(* IEC 61131-3 sources: programs/VI-54/VI-54_20171205/VI-54_20171205/Stations/Screen/LseClass170718/Class/TCPComSend, 1 file *)

(* ---- TCPComSend.st ---- *)
(*!
<Class
	Name               = "TCPComSend"
	Revision           = "1.2"
	RealtimeTask       = "false"
	CyclicTask         = "true"
	BackgroundTask     = "true"
	Sigmatek           = "true"
	OSInterface        = "false"
	HighPriority       = "false"
	Automatic          = "false"
	UpdateMode         = "Prescan"
	SharedCommandTable = "true"
	Objectsize         = "(600,360)"
	Comment            = "Sending data via communication class.">
	<Channels>
		<Server Name="ClassSvr" Visualized="false" Initialize="false" WriteProtected="false" Retentive="false"/>
		<Server Name="ID_Destination" Visualized="false" Initialize="true" WriteProtected="true" Retentive="false"/>
		<Server Name="ID_Source" Visualized="false" Initialize="true" WriteProtected="true" Retentive="false"/>
		<Server Name="sSendCnt" Visualized="false" Initialize="false" WriteProtected="false" Retentive="false" Comment="Counter for sended data blocks."/>
		<Server Name="sSendErr" Visualized="false" Initialize="false" WriteProtected="false" Retentive="false" Comment="Counter for send errors."/>
		<Client Name="cPrio" Required="true" Internal="false" Comment="Communication priority number."/>
		<Client Name="cSendErr" Required="false" Internal="false" Comment="Write out JobID if sending was not Ok."/>
		<Client Name="cSendOk" Required="false" Internal="false" Comment="Write out JobID if sending was Ok."/>
		<Client Name="toDataManager" Required="true" Internal="false" Comment="Connection to communication data manager."/>
	</Channels>
	<RevDoku>
		<Owner Company="Sigmatek GmbH &amp; Co KG" Author="LeiChr"/>
		<Dokumentation Revision="1.2" Date="2015-11-16" Author="HubChr" Company="Sigmatek GmbH &amp; Co KG" Description="Translated error messages of SendData method"/>
		<Dokumentation Revision="1.1" Date="2015-11-11" Author="hötant" Company="Sigmatek GmbH &amp; Co KG" Description="corrected error in SendData method. ( OptCmd did not work )"/>
		<Dokumentation Revision="1.0" Date="2015-07-30" Author="LeiChr" Company="Sigmatek GmbH &amp; Co KG" Description="Initial library version"/>
	</RevDoku>
</Class>
*)
TCPComSend : CLASS
  //Servers:
	ClassSvr 	: SvrChCmd_DINT;
	ID_Destination 	: SvrCh_DINT;
	ID_Source 	: SvrCh_DINT;
	sSendCnt 	: SvrCh_DINT;
	sSendErr 	: SvrCh_DINT;
  //Clients:
	toDataManager 	: CltChCmd_DataManager;
	cPrio 	: CltCh_DINT;
	cSendOk 	: CltCh_DINT;
	cSendErr 	: CltCh_DINT;
  //Variables:
  //Functions:

	FUNCTION VIRTUAL GLOBAL Init;

	FUNCTION VIRTUAL GLOBAL CyWork
		VAR_INPUT
			EAX 	: UDINT;
		END_VAR
		VAR_OUTPUT
			state (EAX) 	: UDINT;
		END_VAR;

	FUNCTION VIRTUAL GLOBAL Background
		VAR_INPUT
			EAX 	: UDINT;
		END_VAR
		VAR_OUTPUT
			state (EAX) 	: UDINT;
		END_VAR;
				//! <Function Comment="Is called everytime the state of a job is changing. Overwrite to react to state changes." Name="CallBackJobState"/>
	FUNCTION VIRTUAL GLOBAL CallBackJobState
		VAR_INPUT
			JobID 	: DINT;
			JobState 	: DataManagerPriority::t_e_CallbackState;
		END_VAR;
				//! <Function Comment="Sends the data" Name="SendData"/>
	FUNCTION VIRTUAL GLOBAL SendData
		VAR_INPUT
			pData 	: ^void;			//! <Variable Comment="Pointer to the data to be sent." Name="SendData.pData"/>
			length 	: UDINT;			//! <Variable Comment="Length of the data to be sent." Name="SendData.length"/>
			timeout 	: UDINT;			//! <Variable Comment="TCP Timeout." Name="SendData.timeout"/>
			OptCMD 	: USINT := 0;			//! <Variable Comment="An optional command value can be set here. In order to receive the command parameter correctly, the method CallBackReciverCMD has to be used." Name="SendData.OptCMD"/>
		END_VAR
		VAR_OUTPUT
			JobID 	: DINT;			//! <Variable Comment="ID of the job." Name="SendData.JobID"/>
		END_VAR;
  //Tables:
	FUNCTION @STD
		VAR_OUTPUT
			ret_code	: CONFSTATES;
		END_VAR;
	FUNCTION GLOBAL TAB @CT_;
END_CLASS;

#pragma usingLtd DataManager

// ********************************************************************
// Prototype of callbackmethod
// ********************************************************************
// ********************************************************************
FUNCTION GLOBAL Com_SendData_Callback
	VAR_INPUT
		pthis 	: ^void;
		JobID 	: DINT;
		JobState 	: DataManagerPriority::t_e_CallbackState;
	END_VAR

  pthis$^TCPComSend^.CallBackJobState(JobID, JobState);

END_FUNCTION

// ********************************************************************
// Init
// ********************************************************************
// ********************************************************************
FUNCTION VIRTUAL GLOBAL TCPComSend::Init

  if _FirstScan then
  end_if;

END_FUNCTION

// ********************************************************************
// Callbackmethod of send
// ********************************************************************
// ********************************************************************
FUNCTION VIRTUAL GLOBAL TCPComSend::CallBackJobState
	VAR_INPUT
		JobID 	: DINT;
		JobState 	: DataManagerPriority::t_e_CallbackState;
	END_VAR

  case JobState of
    //Ok
    _MNG_Received:
       cSendOk :=JobID;
       cSendOk.write (cSendOk);

    //Error
    _MNG_NoReceiverConnected,
    _MNG_GlobalReceiveError,
    _MNG_TimeOut:
       cSendErr :=JobId;
       cSendErr.write (cSendErr);
       sSendErr +=1;
  end_case;

END_FUNCTION

// ********************************************************************
// Sendmethod
// ********************************************************************
// ********************************************************************
FUNCTION VIRTUAL GLOBAL TCPComSend::SendData
	VAR_INPUT
		pData 	: ^void;
		length 	: UDINT;
		timeout 	: UDINT;
		OptCMD 	: USINT;
	END_VAR
	VAR_OUTPUT
		JobID 	: DINT;
	END_VAR
  VAR
  	tmpDestinationID: DINT;
    txt1 : array [0..199] of char;
    txt2 : array [0..99] of char;
    txtOut : array [0..599] of char;
  END_VAR

  tmpDestinationID := to_dint(OptCMD);
  tmpDestinationID := tmpDestinationID shl 24;
  tmpDestinationID := tmpDestinationID OR ( ID_Destination AND 16#00FFFFFF );

  cPrio := cPrio.Read();
  Jobid := toDataManager.SetData(  tmpDestinationID,
                              ID_Source,
                              pData,
                              length,
                              this,
                              #Com_SendData_Callback(),
                              timeout,
                              cPrio);

  if JobID <0 then
    sSendErr +=1;
    case JobID of
      -1 :  _strcpy(dest:=#txt1[0], src:="Buffer Problem!");
      -2 :  _strcpy(dest:=#txt1[0], src:="Offline!");
      -3 :  _strcpy(dest:=#txt1[0], src:="Invalid Priority!");
      -4 :  _strcpy(dest:=#txt1[0], src:="Method may not be called from RtWork!");
    else
      _strcpy(dest:=#txt1[0], src:="Unknown return value");
    end_case;
    _GetObjName(pThis:=this, pName:=#txt2[0]);
    _strcpy(dest:=#txtout[0], src:=#txt2[0]);
    _strcat(dest:=#txtout[0], src:="-> SendData -> ");
    _strcat(dest:=#txtout[0], src:=#txt1[0]);
    TRACE(#txtout[0]);
  else
    sSendCnt +=1;
  end_if;

END_FUNCTION

// ********************************************************************
// cywork
// ********************************************************************
// ********************************************************************
FUNCTION VIRTUAL GLOBAL TCPComSend::CyWork
	VAR_INPUT
		EAX 	: UDINT;
	END_VAR
	VAR_OUTPUT
		state (EAX) 	: UDINT;
	END_VAR

	state := READY;

END_FUNCTION

// ********************************************************************
// Background
// ********************************************************************
// ********************************************************************
FUNCTION VIRTUAL GLOBAL TCPComSend::Background
	VAR_INPUT
		EAX 	: UDINT;
	END_VAR
	VAR_OUTPUT
		state (EAX) 	: UDINT;
	END_VAR

	state := READY;

END_FUNCTION
